IF bIX_TriplexRPMAutoMode = 0 OR bTriplexRPMEnable  = 0 (*Если переключен в режим "Ручной" извне переключателем или отключен с дисплея, то ПИД отключаем*)
THEN
	PID_2_Reset    := 1;
	(*rSet_GN2Rate   := 0;  ЗАЧЕМ!!!!!!!!!!!!!!!!!!!*)
	PID_2_Y_Manual := 1;
ELSE
	PID_2_Reset    := 0;
	PID_2_Y_Manual := 0;
END_IF;

(*-----------------------------------------------------------------------------------------------------------------------------------------------------------------------------------*)
(*Ограничиваем устанавливаемое максимальное значение оборотов*)

IF rSet_TriplexRPM > 975 THEN
	rSet_TriplexRPM := 975;
END_IF;

(*-----------------------------------------------------------------------------------------------------------------------------------------------------------------------------------*)
(*ПИД-контур 1 поддержания скорости НВД*)

PID_2(Actual      := rFRQ_TriplexRPM,
	Set_Point     := rSet_TriplexRPM,
	KP            := rArrayDataPID_P_Coef[2],
	TN            := rArrayDataPID_I_Coef[2],
	TV            := rArrayDataPID_D_Coef[2],
	Y_Manual      := PID_2_Y_Manual,
	Y_Offset      := rArrayDataPID_Shift[2],
	Y_Min         := rArrayDataPWM_YL[2],
	Y_Max         := rArrayDataPWM_YH[2] (*PID_2_Y_Max*),
	Manual        := PID_2_Manual,
	Reset         := PID_2_Reset,
	Y             => rPWM_TriplexRPM,
	Limits_Active => PID_2_Limits,
	Overflow      => PID_2_Overflow);

rArrayDataRAWPID[2] := rPWM_TriplexRPM;

(*-----------------------------------------------------------------------------------------------------------------------------------------------------------------------------------*)
(*Отключаемся от управления ШИМ в режиме "Ручной"*)

IF bIX_TriplexRPMAutoMode = 0 OR bTriplexRPMEnable  = 0 (*Если переключен в режим "Ручной" извне переключателем или отключен с дисплея, то ШИМ отключаем*)
THEN
	rPWM_TriplexRPM := 0;
END_IF;

(*-----------------------------------------------------------------------------------------------------------------------------------------------------------------------------------*)
(*Обработка байта описания канала*)

CASE dwArrayDataPWM_DZ_MIN[2] OF
	0: rPWM_TriplexRPM := rPWM_TriplexRPM;
	1: rPWM_TriplexRPM := rArrayDataPWM_DZ_MAX[2];
	2: rPWM_TriplexRPM := rPWM_TriplexRPM * rArrayDataPWM_DZ_MAX[2];
	ELSE rPWM_TriplexRPM := rPWM_TriplexRPM;
END_CASE;

rArrayDataRAWPWM[2] := rPWM_TriplexRPM;

(*-----------------------------------------------------------------------------------------------------------------------------------------------------------------------------------*)
(*ШИМ-контроллер поддержания скорости НВД*)

TriplexRPMFreqPWM(dwReriodPWM := dwArrayAverTimePWM[2], wFrequencyPWM => , bRestartPWM => );

PWM2(INIT := (bFirstIn OR TriplexRPMFreqPWM.bRestartPWM), FREQUENCY := TriplexRPMFreqPWM.wFrequencyPWM, CHANNEL := 1, VALUE := REAL_TO_WORD(rPWM_TriplexRPM), CHANGE := TRUE, DITHER_VALUE := 10, DITHER_FREQUENCY := 140);

(*-----------------------------------------------------------------------------------------------------------------------------------------------------------------------------------*)
(**)

bIX_TriplexRPMAutoModePrev := bIX_TriplexRPMAutoMode;

(*-----------------------------------------------------------------------------------------------------------------------------------------------------------------------------------*)
(*Расчет рассогласования расчетной и текущей величины*)

rTriplexRPM_Calc := TriplexRPM_calculation(rPWMcurr := (rPWM_TriplexRPM / 10), rRPMeng := DINT_TO_REAL(diCurrentEngineRPM));

IF rFRQ_TriplexRPM > 1
THEN
	rTriplexRPM_Err := (rTriplexRPM_Calc - rFRQ_TriplexRPM) * 100 / rFRQ_TriplexRPM;
ELSE
	rTriplexRPM_Err := 0;
END_IF;

(*-----------------------------------------------------------------------------------------------------------------------------------------------------------------------------------*)
(*bErrorNumber16 - Ошибка 16. НВД. Переведите регулятор в положение «0»*)
(*
IF byCurrStep = 3 AND bTriplexRPMEnable = 1 AND ABS(rTriplexRPM_Err) > 20
THEN
	bErrorNumber16  := 1;(*РАБОТАЕМ С ПРЕДУПРЕЖДЕНИЕМ*)
	dwHornEnable.16 := 0;(*Сирена отключена*)
ELSE
	bErrorNumber16  := 0;
	dwHornEnable.16 := 0;
END_IF;*)
END_PROGRAM

(* POU Service/Temperature_calculation, ST *)
FUNCTION Temperature_calculation : REAL (*Tемпература предварительного прогрева*)

VAR_INPUT
	rTmin : REAL := 0;(*Минимальная температура прогрева, C*)
	rVreq : REAL := 0;(*Заданный расход газообразного азота, м3/мин*)
	rPprs : REAL := 0;(*Давление нагнетания, Мпа*)
	rTreq : REAL := 0;(*Заданная температура нагнетания, С*)
	rK    : REAL := 0;(*Коэффициент теплопередачи*)
END_VAR

VAR
	rTadd : REAL := 0;(*Дополнительная температура подогрева связанная с расходом, C*)
END_VAR
(*-----------------------------------------------------------------------------------------------------------------------------------------------------------------------------------*)
(**)

IF rPprs > 0.1
THEN
	rTadd := 1.8741643E-5 * rVreq * (11760 - 86.5 * SQRT(10 * rPprs - 1) + 0.0255 * (EXPT((rTreq + 273.15), 2) - EXPT(293.15, 2)));
ELSE
	rTadd := 1.8741643E-5 * rVreq * (11760 - 86.5 * SQRT(10 * 0.1 - 1) + 0.0255 * (EXPT((rTreq + 273.15), 2) - EXPT(293.15, 2)));
END_IF;

Temperature_calculation := rTmin + rTadd;
END_FUNCTION

(* POU Service/TriplexRPM_calculation, ST *)
FUNCTION TriplexRPM_calculation : REAL (*Расчетное значение оборотов НВД, об/мин*)

VAR_INPUT
	rPWMcurr : REAL;(*Текущее значение ШИМ, %*)
	rRPMeng  : REAL;(*Обороты двигателя, об/мин*)
END_VAR

VAR
END_VAR
(*-----------------------------------------------------------------------------------------------------------------------------------------------------------------------------------*)
(**)

TriplexRPM_calculation := 0.002187 * rRPMeng * (10 * rPWMcurr - rArrayDataPID_Shift[2]);
END_FUNCTION

(* POU ChannelCalc_processing, ST *)
PROGRAM ChannelCalc_processing

VAR_INPUT
	bInit             : BOOL;
END_VAR

VAR
	AIN_processing_00 : Linearization_AIN_processing;
	AIN_processing_01 : Linearization_AIN_processing;

	AIN_processing_03 : Linearization_AIN_processing;
	AIN_processing_04 : Linearization_AIN_processing;
	AIN_processing_05 : Linearization_AIN_processing;

	AIN_processing_08 : Linearization_AIN_processing;

	PIN_processing_00 : Linearization_PIN_processing;

	PWM_processing_00 : Extraction_PWM_processing;
	PWM_processing_01 : Extraction_PWM_processing;
	PWM_processing_02 : Extraction_PWM_processing;

	PID_processing_00 : Extraction_PID_processing;
	PID_processing_01 : Extraction_PID_processing;
	PID_processing_02 : Extraction_PID_processing;

	i                 : INT := 0;
END_VAR
(*-----------------------------------------------------------------------------------------------------------------------------------------------------------------------------------*)
(**)

FOR i := 0 TO 63 DO

	IF aPage_Channel[i].PARAM_00 = 0
	THEN
		aPage_Channel[i].PARAM_08 := rArrayDataRAWADC[aPage_Channel[i].PARAM_09];
	END_IF;

	IF aPage_Channel[i].PARAM_00 = 1
	THEN
		aPage_Channel[i].PARAM_08 := rArrayDataRAWPIN[aPage_Channel[i].PARAM_09];
	END_IF;

	IF aPage_Channel[i].PARAM_00 = 2
	THEN
		aPage_Channel[i].PARAM_08 := rArrayDataRAWPWM[aPage_Channel[i].PARAM_09];
	END_IF;

	IF aPage_Channel[i].PARAM_00 = 3
	THEN
		aPage_Channel[i].PARAM_08 := rArrayDataRAWPID[aPage_Channel[i].PARAM_09];
	END_IF;

END_FOR;

(*-----------------------------------------------------------------------------------------------------------------------------------------------------------------------------------*)
(**)

AIN_processing_00(
	Page_Channel_AIN := aPage_Channel[0],
	rADC_ValueHigh   := rADC_ValueHigh,
	rADC_ValueLow    := rADC_ValueLow,
	sParamName       => ,
	rOutputValue     => rIW_BoostPres,
	bErrADC_Value    => bErrorBoostPres,
	bErrInputValue   => );

AIN_processing_01(
	Page_Channel_AIN := aPage_Channel[1],
	rADC_ValueHigh   := rADC_ValueHigh,
	rADC_ValueLow    := rADC_ValueLow,
	sParamName       => ,
	rOutputValue     => rIW_LN2_Temp,
	bErrADC_Value    => bErrorLN2_Temp,
	bErrInputValue   => );

AIN_processing_03(
	Page_Channel_AIN := aPage_Channel[2],
	rADC_ValueHigh   := rADC_ValueHigh,
	rADC_ValueLow    := rADC_ValueLow,
	sParamName       => ,
	rOutputValue     => rIW_GN2_Temp,
	bErrADC_Value    => bErrorGN2_Temp,
	bErrInputValue   => );

AIN_processing_04(
	Page_Channel_AIN := aPage_Channel[3],
	rADC_ValueHigh   := rADC_ValueHigh,
	rADC_ValueLow    := rADC_ValueLow,
	sParamName       => ,
	rOutputValue     => rIW_GN2_Pres,
	bErrADC_Value    => bErrorGN2_Pres,
	bErrInputValue   => );

AIN_processing_05(
	Page_Channel_AIN := aPage_Channel[4],
	rADC_ValueHigh   := rADC_ValueHigh,
	rADC_ValueLow    := rADC_ValueLow,
	sParamName       => ,
	rOutputValue     => rIW_HydHeatPres,
	bErrADC_Value    => bErrorHydHeatPres,
	bErrInputValue   => );

AIN_processing_08(
	Page_Channel_AIN := aPage_Channel[5],
	rADC_ValueHigh   := rADC_ValueHigh,
	rADC_ValueLow    := rADC_ValueLow,
	sParamName       => ,
	rOutputValue     => rIW_CoolTempIn,
	bErrADC_Value    => bErrorCoolTempIn,
	bErrInputValue   => );

(*-----------------------------------------------------------------------------------------------------------------------------------------------------------------------------------*)
(**)

PIN_processing_00(
	Page_Channel_PIN := aPage_Channel[6],
	rFRQ_ValueHigh   := 10_000,
	rFRQ_ValueLow    := -1,
	sParamName       => ,
	rOutputValue     => rFRQ_TriplexRPM,
	bErrFRQ_Value    => ,
	bErrInputValue   => );

IF diCurrentEngineRPM < 500
THEN
	rFRQ_TriplexRPM := 0;
END_IF;

(*-----------------------------------------------------------------------------------------------------------------------------------------------------------------------------------*)
(**)

PWM_processing_00(
	Page_Channel_PWM := aPage_Channel[7],
	sParamName       =>,
	rDataPWM_XH      => rArrayDataPWM_XH[1],
	rDataPWM_XL      => rArrayDataPWM_XL[1],
	rDataPWM_YH      => rArrayDataPWM_YH[1],
	rDataPWM_YL      => rArrayDataPWM_YL[1],
	dwAverTimePWM    => dwArrayAverTimePWM[1],
	rDataPWM_DZ_MAX  => rArrayDataPWM_DZ_MAX[1],
	dwDataPWM_DZ_MIN => dwArrayDataPWM_DZ_MIN[1],
	dwNumberPWM      => dwArrayNumberPWM[1],
	rParam10PWM      => rArrayParam10PWM[1]);

PWM_processing_01(
	Page_Channel_PWM := aPage_Channel[8],
	sParamName       =>,
	rDataPWM_XH      => rArrayDataPWM_XH[2],
	rDataPWM_XL      => rArrayDataPWM_XL[2],
	rDataPWM_YH      => rArrayDataPWM_YH[2],
	rDataPWM_YL      => rArrayDataPWM_YL[2],
	dwAverTimePWM    => dwArrayAverTimePWM[2],
	rDataPWM_DZ_MAX  => rArrayDataPWM_DZ_MAX[2],
	dwDataPWM_DZ_MIN => dwArrayDataPWM_DZ_MIN[2],
	dwNumberPWM      => dwArrayNumberPWM[2],
	rParam10PWM      => rArrayParam10PWM[2]);

PWM_processing_02(
	Page_Channel_PWM := aPage_Channel[9],
	sParamName       =>,
	rDataPWM_XH      => rArrayDataPWM_XH[3],
	rDataPWM_XL      => rArrayDataPWM_XL[3],
	rDataPWM_YH      => rArrayDataPWM_YH[3],
	rDataPWM_YL      => rArrayDataPWM_YL[3],
	dwAverTimePWM    => dwArrayAverTimePWM[3],
	rDataPWM_DZ_MAX  => rArrayDataPWM_DZ_MAX[3],
	dwDataPWM_DZ_MIN => dwArrayDataPWM_DZ_MIN[3],
	dwNumberPWM      => dwArrayNumberPWM[3],
	rParam10PWM      => rArrayParam10PWM[3]);

(*-----------------------------------------------------------------------------------------------------------------------------------------------------------------------------------*)
(**)

PID_processing_00(
	Page_Channel_PID := aPage_Channel[10],
	sParamName       =>,
	rDataPID_P_Coef  => rArrayDataPID_P_Coef[1],
	rDataPID_I_Coef  => rArrayDataPID_I_Coef[1],
	rDataPID_D_Coef  => rArrayDataPID_D_Coef[1],
	rDataPID_Shift   => rArrayDataPID_Shift[1],
	dwAverTimePID    => dwArrayAverTimePID[1],
	rCoeffPID        => rArrayCoeffPID[1],
	dwDescriptPID    => dwArrayDescriptPID[1],
	dwNumberPID      => dwArrayNumberPID[1],
	rParam10PID      => rArrayParam10PID[1]);

PID_processing_01(
	Page_Channel_PID := aPage_Channel[11],
	sParamName       =>,
	rDataPID_P_Coef  => rArrayDataPID_P_Coef[2],
	rDataPID_I_Coef  => rArrayDataPID_I_Coef[2],
	rDataPID_D_Coef  => rArrayDataPID_D_Coef[2],
	rDataPID_Shift   => rArrayDataPID_Shift[2],
	dwAverTimePID    => dwArrayAverTimePID[2],
	rCoeffPID        => rArrayCoeffPID[2],
	dwDescriptPID    => dwArrayDescriptPID[2],
	dwNumberPID      => dwArrayNumberPID[2],
	rParam10PID      => rArrayParam10PID[2]);

PID_processing_02(
	Page_Channel_PID := aPage_Channel[12],
	sParamName       =>,
	rDataPID_P_Coef  => rArrayDataPID_P_Coef[3],
	rDataPID_I_Coef  => rArrayDataPID_I_Coef[3],
	rDataPID_D_Coef  => rArrayDataPID_D_Coef[3],
	rDataPID_Shift   => rArrayDataPID_Shift[3],
	dwAverTimePID    => dwArrayAverTimePID[3],
	rCoeffPID        => rArrayCoeffPID[3],
	dwDescriptPID    => dwArrayDescriptPID[3],
	dwNumberPID      => dwArrayNumberPID[3],
	rParam10PID      => rArrayParam10PID[3]);

(*-----------------------------------------------------------------------------------------------------------------------------------------------------------------------------------*)
(**)

bCommomErrorADC := (bErrorBoostPres OR
					bErrorLN2_Temp OR
					bErrorGN2_Temp OR
					bErrorGN2_Pres OR
					(*bErrorHydHeatPres OR*)
					bErrorCoolTempIn);

(*-----------------------------------------------------------------------------------------------------------------------------------------------------------------------------------*)
(*Расчет текущей производительности установки*)

IF rFRQ_TriplexRPM > 0
THEN
	rCurrent_GN2Rate := 0.08786324786325 * rFRQ_TriplexRPM; (*м3/оборот * оборот/мин*)
ELSE
	rCurrent_GN2Rate := 0;
END_IF;

udiCurrent_GN2RateLitres := REAL_TO_DWORD(rCurrent_GN2Rate * 1000);

(*-----------------------------------------------------------------------------------------------------------------------------------------------------------------------------------*)
(**)
END_PROGRAM

(* POU Linearization_AIN_processing, ST *)
FUNCTION_BLOCK Linearization_AIN_processing

VAR_INPUT
	Page_Channel_AIN  : Page_Channel;
	rADC_ValueHigh    : REAL;
	rADC_ValueLow     : REAL;
END_VAR

VAR_OUTPUT
	sParamName        : STRING(32);
	rOutputValue      : REAL := 0;
	bErrADC_Value     : BOOL := 0;
	bErrInputValue    : BOOL := 0;
END_VAR

VAR
	rArrayDataADC     : ARRAY [0..257] OF REAL;(*Массив необработанных данных канала, REAL*)
	rTotalADC         : REAL := 0;(**)
	iIndexReadings    : INT  := 0;(**)
	diNumReadings     : DINT := 10;(*Рассчитанное число измерений для усреднения*)
	diNumReadingsPrev : DINT := 0;
	rDataOutADC       : REAL;(*Усредненное значение канала*)
	i                 : INT  := 0;

	bErrADC_ValueHigh : BOOL := 0;
	bErrADC_ValueLow  : BOOL := 0;
END_VAR
(*-----------------------------------------------------------------------------------------------------------------------------------------------------------------------------------*)
(**)

sParamName := Page_Channel_AIN.PARAM_NAME;

(*-----------------------------------------------------------------------------------------------------------------------------------------------------------------------------------*)
(*Усредняем значене канала*)

diNumReadings := (DWORD_TO_DINT(Page_Channel_AIN.PARAM_05) * 1000) / 10_000 (*DWORD_TO_DINT(dwCycleTime)*);(**)
IF diNumReadings < 1   THEN diNumReadings := 1;   END_IF;
IF diNumReadings > 255 THEN diNumReadings := 255; END_IF;

IF diNumReadings <> diNumReadingsPrev
THEN
	rTotalADC := 0;
	FOR i := 1 TO DINT_TO_INT(diNumReadings) DO
	rTotalADC := rTotalADC + rArrayDataADC[i - 1];
	END_FOR;
END_IF;

diNumReadingsPrev := diNumReadings;

rTotalADC := rTotalADC - rArrayDataADC[iIndexReadings];(*subtract the last reading*)

rArrayDataADC[iIndexReadings] := Page_Channel_AIN.PARAM_08;(*read from the sensor*)

rTotalADC := rTotalADC + rArrayDataADC[iIndexReadings];(*add the reading to the total*)

iIndexReadings := iIndexReadings + 1;(*advance to the next position in the array*)

IF INT_TO_DINT(iIndexReadings) >= diNumReadings THEN iIndexReadings := 0; END_IF;(*if we're at the end of the array... ...wrap around to the beginning*)

rDataOutADC := rTotalADC / DINT_TO_REAL(diNumReadings);(**)

(*-----------------------------------------------------------------------------------------------------------------------------------------------------------------------------------*)
(*Основная обработка аналогового канала*)

(*Обработка обрывов (значение меньше минимально допустимого) и КЗ (значение больше максимально допустимого) по входу канала*)
IF rDataOutADC > rADC_ValueHigh
THEN bErrADC_ValueHigh := 1;
ELSE bErrADC_ValueHigh := 0;
END_IF;

IF rDataOutADC < rADC_ValueLow
THEN bErrADC_ValueLow := 1;
ELSE bErrADC_ValueLow := 0;
END_IF;

bErrADC_Value := bErrADC_ValueHigh OR bErrADC_ValueLow;

(*Масштабирование значений каналов*)
IF Page_Channel_AIN.PARAM_01 = Page_Channel_AIN.PARAM_02
THEN
	rOutputValue := rDataOutADC;(*Защита от деления на 0, выводим необработанные значения АЦП*)
	bErrInputValue := 1;
ELSE
	rOutputValue := (Page_Channel_AIN.PARAM_03 - Page_Channel_AIN.PARAM_04) / (Page_Channel_AIN.PARAM_01 - Page_Channel_AIN.PARAM_02) * rDataOutADC + (Page_Channel_AIN.PARAM_04 - (Page_Channel_AIN.PARAM_03 - Page_Channel_AIN.PARAM_04) / (Page_Channel_AIN.PARAM_01 - Page_Channel_AIN.PARAM_02) * Page_Channel_AIN.PARAM_02);
	bErrInputValue := 0;
END_IF;

(*Обработка байта описания канала*)
CASE Page_Channel_AIN.PARAM_07 OF
	0: rOutputValue := rOutputValue;
	1: rOutputValue := Page_Channel_AIN.PARAM_06;
	2: rOutputValue := rOutputValue * Page_Channel_AIN.PARAM_06;
ELSE
	rOutputValue := rOutputValue;
END_CASE;

(*Если обнаружена ошибка по каналу, то подставляем заведомо неверное число*)
	IF bErrADC_Value = 1 OR bErrInputValue = 1 THEN rOutputValue := -9999; END_IF;

(*-----------------------------------------------------------------------------------------------------------------------------------------------------------------------------------*)
(**)
END_FUNCTION_BLOCK

(* POU Linearization_PIN_processing, ST *)
FUNCTION_BLOCK Linearization_PIN_processing

VAR_INPUT
	Page_Channel_PIN  : Page_Channel;
	rFRQ_ValueHigh    : REAL;
	rFRQ_ValueLow     : REAL;
END_VAR

VAR_OUTPUT
	sParamName        : STRING(32);
	rOutputValue      : REAL := 0;
	bErrFRQ_Value     : BOOL := 0;
	bErrInputValue    : BOOL := 0;
END_VAR

VAR
	rArrayDataFRQ     : ARRAY [0..257] OF REAL;(*Массив необработанных данных канала, REAL*)
	rTotalFRQ         : REAL := 0;(**)
	rTotalFRQ2        : REAL := 0;(**)
	iIndexReadings    : INT  := 0;(**)
	diNumReadings     : DINT := 10;(*Рассчитанное число измерений для усреднения*)
	diNumReadingsPrev : DINT := 0;
	rDataOutFRQ       : REAL;(*Усредненное значение канала*)
	i                 : INT  := 0;

	bErrFRQ_ValueHigh : BOOL := 0;
	bErrFRQ_ValueLow  : BOOL := 0;
END_VAR
(*-----------------------------------------------------------------------------------------------------------------------------------------------------------------------------------*)
(**)

sParamName := Page_Channel_PIN.PARAM_NAME;

(*-----------------------------------------------------------------------------------------------------------------------------------------------------------------------------------*)
(*Усредняем значене канала*)

diNumReadings := (DWORD_TO_DINT(Page_Channel_PIN.PARAM_05) * 1000) / 10_000 (*DWORD_TO_DINT(dwCycleTime)*);(**)
IF diNumReadings < 1   THEN diNumReadings := 1;   END_IF;
IF diNumReadings > 255 THEN diNumReadings := 255; END_IF;

IF diNumReadings <> diNumReadingsPrev
THEN
	rTotalFRQ  := 0;
	rTotalFRQ2 := 0;
	FOR i := 1 TO DINT_TO_INT(diNumReadings) DO
	rTotalFRQ  := rTotalFRQ  + rArrayDataFRQ[i - 1];
	rTotalFRQ2 := rTotalFRQ;
	END_FOR;
END_IF;

diNumReadingsPrev := diNumReadings;

rTotalFRQ := rTotalFRQ - rArrayDataFRQ[iIndexReadings];(*subtract the last reading*)

rArrayDataFRQ[iIndexReadings] := Page_Channel_PIN.PARAM_08;(*read from the sensor*)

rTotalFRQ := rTotalFRQ + rArrayDataFRQ[iIndexReadings];(*add the reading to the total*)

rTotalFRQ2 := rTotalFRQ2 + rArrayDataFRQ[iIndexReadings];

iIndexReadings := iIndexReadings + 1;(*advance to the next position in the array*)

IF INT_TO_DINT(iIndexReadings) >= diNumReadings
THEN
	IF rTotalFRQ2 < 1
	THEN rTotalFRQ := 0;
	END_IF;
END_IF;

IF INT_TO_DINT(iIndexReadings) >= diNumReadings THEN iIndexReadings := 0; rTotalFRQ2 := 0; END_IF;(*if we're at the end of the array... ...wrap around to the beginning*)

rDataOutFRQ := rTotalFRQ / DINT_TO_REAL(diNumReadings);(**)

(*-----------------------------------------------------------------------------------------------------------------------------------------------------------------------------------*)
(*Основная обработка частотного канала*)

(*Обработка ошибочных частот (значение меньше минимально допустимого и значение больше максимально допустимого) по входу канала*)
IF rDataOutFRQ > rFRQ_ValueHigh
THEN bErrFRQ_ValueHigh := 1;
ELSE bErrFRQ_ValueHigh := 0;
END_IF;

IF rDataOutFRQ < rFRQ_ValueLow
THEN bErrFRQ_ValueLow := 1;
ELSE bErrFRQ_ValueLow := 0;
END_IF;

bErrFRQ_Value := bErrFRQ_ValueHigh OR bErrFRQ_ValueLow;

(*Масштабирование значений каналов*)
IF Page_Channel_PIN.PARAM_01 = Page_Channel_PIN.PARAM_02
THEN
	rOutputValue := rDataOutFRQ;(*Защита от деления на 0, выводим необработанные значения частоты*)
	bErrInputValue := 1;
ELSE
	rOutputValue := (Page_Channel_PIN.PARAM_03 - Page_Channel_PIN.PARAM_04) / (Page_Channel_PIN.PARAM_01 - Page_Channel_PIN.PARAM_02) * rDataOutFRQ;
	bErrInputValue := 0;
END_IF;

(*Обработка байта описания канала*)
CASE Page_Channel_PIN.PARAM_07 OF
	0: rOutputValue := rOutputValue;
	1: rOutputValue := Page_Channel_PIN.PARAM_06;
	2: rOutputValue := rOutputValue * Page_Channel_PIN.PARAM_06;
ELSE
	rOutputValue := rOutputValue;
END_CASE;

(*Если обнаружена ошибка по каналу, то подставляем заведомо неверное число*)
	IF bErrFRQ_Value = 1 OR bErrInputValue = 1 THEN rOutputValue := -9999; END_IF;

(*-----------------------------------------------------------------------------------------------------------------------------------------------------------------------------------*)
(**)
END_FUNCTION_BLOCK

(* POU Extraction_PWM_processing, ST *)
FUNCTION_BLOCK Extraction_PWM_processing

VAR_INPUT
	Page_Channel_PWM : Page_Channel;
END_VAR

VAR_OUTPUT
	sParamName       : STRING(32);
	rDataPWM_XH      : REAL;
	rDataPWM_XL      : REAL;
	rDataPWM_YH      : REAL;
	rDataPWM_YL      : REAL;
	dwAverTimePWM    : DWORD;
	rDataPWM_DZ_MAX  : REAL;
	dwDataPWM_DZ_MIN : DWORD;
	dwNumberPWM      : DWORD;
	rParam10PWM      : REAL;
END_VAR

VAR
END_VAR
(*-----------------------------------------------------------------------------------------------------------------------------------------------------------------------------------*)
(**)

sParamName       := Page_Channel_PWM.PARAM_NAME;
rDataPWM_XH      := Page_Channel_PWM.PARAM_01;
rDataPWM_XL      := Page_Channel_PWM.PARAM_02;
rDataPWM_YH      := Page_Channel_PWM.PARAM_03;
rDataPWM_YL      := Page_Channel_PWM.PARAM_04;
dwAverTimePWM    := Page_Channel_PWM.PARAM_05;
rDataPWM_DZ_MAX  := Page_Channel_PWM.PARAM_06;
dwDataPWM_DZ_MIN := Page_Channel_PWM.PARAM_07;

dwNumberPWM      := Page_Channel_PWM.PARAM_09;
rParam10PWM      := Page_Channel_PWM.PARAM_10;
END_FUNCTION_BLOCK

(* POU Extraction_PID_processing, ST *)
FUNCTION_BLOCK Extraction_PID_processing

VAR_INPUT
	Page_Channel_PID : Page_Channel;
END_VAR

VAR_OUTPUT
	sParamName      : STRING(32);
	rDataPID_P_Coef : REAL;
	rDataPID_I_Coef : REAL;
	rDataPID_D_Coef : REAL;
	rDataPID_Shift  : REAL;
	dwAverTimePID   : DWORD;
	rCoeffPID       : REAL;
	dwDescriptPID   : DWORD;
	dwNumberPID     : DWORD;
	rParam10PID     : REAL;
END_VAR

VAR
END_VAR
(*-----------------------------------------------------------------------------------------------------------------------------------------------------------------------------------*)
(**)

sParamName      := Page_Channel_PID.PARAM_NAME;
rDataPID_P_Coef := Page_Channel_PID.PARAM_01;
rDataPID_I_Coef := Page_Channel_PID.PARAM_02;
rDataPID_D_Coef := Page_Channel_PID.PARAM_03;
rDataPID_Shift  := Page_Channel_PID.PARAM_04;
dwAverTimePID   := Page_Channel_PID.PARAM_05;
rCoeffPID       := Page_Channel_PID.PARAM_06;
dwDescriptPID   := Page_Channel_PID.PARAM_07;

dwNumberPID     := Page_Channel_PID.PARAM_09;
rParam10PID     := Page_Channel_PID.PARAM_10;
END_FUNCTION_BLOCK

(* POU Adder_processing, ST *)
PROGRAM Adder_processing

VAR_INPUT
	bInit                    : BOOL;
END_VAR

VAR
	dwTimePrevious           : DWORD := 0;
	dwDeltaTime              : DWORD := 0;

	instFRAMWrite            : FRAMWRITE;
	instFRAMRead             : FRAMREAD;

	i                        : INT;
	k                        : INT;
END_VAR
(*-----------------------------------------------------------------------------------------------------------------------------------------------------------------------------------*)
(*Собираем флаги сброса сумматоров частотных каналов в массив*)

bArrayDataPINAdderReset[1] := bResetTotalAmountGN2 (*bFlowmeterReset_1*);
bArrayDataPINAdderReset[2] := bFlowmeterReset_2;
bArrayDataPINAdderReset[3] := bFlowmeterReset_3;
bArrayDataPINAdderReset[4] := bFlowmeterReset_4;

(*-----------------------------------------------------------------------------------------------------------------------------------------------------------------------------------*)
(*Накопление текущих значений и обработка флагов сброса суммирующих каналов*)

IF k < 100 (*10?*) THEN k := k + 1; ELSE k := 0; END_IF;

IF k = 1
THEN
	dwDeltaTime := (dwTime_US - dwTimePrevious) / 1000;
	FOR i := 1 TO 4 DO
		instFRAMRead(Enable := TRUE, SRC := iMemAdrPINAdder[i], LEN := 4, DST := ADR(udiArrayDataPINAdderOut[i]));(*Извлечение из FRAM значение расходомера i*)

		IF bArrayDataPINAdderReset[i] = 1
			THEN udiArrayDataPINAdderOut[i] := 0;
			ELSE udiArrayDataPINAdderOut[i] := udiArrayDataPINAdderOut[i] + ((udiCurrent_GN2RateLitres * 10 * DWORD_TO_UDINT(dwDeltaTime)) / 60 / 1_000);(*Храним в 0,1 литра*)
		END_IF;

		instFRAMWrite(Enable := TRUE, DST := iMemAdrPINAdder[i], LEN := 4, SRC := ADR(udiArrayDataPINAdderOut[i])); (*Cохранение в FRAM значение расходомера i*)
		END_FOR;

	dwTimePrevious := dwTime_US;

(*-----------------------------------------------------------------------------------------------------------------------------------------------------------------------------------*)
(*Сброс флага "Обнулить накопленное значение расходомера"*)

	bResetTotalAmountGN2 (*bFlowmeterReset_1*) := 0;(*Сброс флага "Обнулить накопленное значение расходомера 0"*)
	bFlowmeterReset_2 := 0;(*Сброс флага "Обнулить накопленное значение расходомера 1"*)
	bFlowmeterReset_3 := 0;(*Сброс флага "Обнулить накопленное значение расходомера 2"*)
	bFlowmeterReset_4 := 0;(*Сброс флага "Обнулить накопленное значение расходомера 3"*)
END_IF;

(*-----------------------------------------------------------------------------------------------------------------------------------------------------------------------------------*)
(*Оформляем необходимые данные для дальнейшей обработки в других блоках*)

rTotalAmountGN2 := UDINT_TO_REAL(udiArrayDataPINAdderOut[1]) / 1000 / 10;
END_PROGRAM

(* POU Output Modules/ProcessState_processing, ST *)
PROGRAM ProcessState_processing

VAR_INPUT
	bFirstIn   : BOOL;
END_VAR

VAR
END_VAR
dwProcessState := 16#0000;

dwProcessState.0 := bDefaultSettings;
dwProcessState.1 := bStop;
dwProcessState.2 := bHornDisable;
dwProcessState.3 := bBlockDisable;

dwProcessState.5 := bIX_BlockOff;

dwProcessState.7 := NOT bQX_TriplexEmergStopTrig;
END_PROGRAM

(* POU Output Modules/Error_processing, ST *)
PROGRAM Error_processing

VAR_INPUT
	bFirstIn            : BOOL;
END_VAR

VAR
	RSInst              : RS;(*Триггер на блокировку*)

	RTRIGInst01         : R_TRIG;
	RTRIGInst02         : R_TRIG;
	RTRIGInst03         : R_TRIG;
	RTRIGInst04         : R_TRIG;
	RTRIGInst05         : R_TRIG;
	RTRIGInst06         : R_TRIG;
	RTRIGInst07         : R_TRIG;
	RTRIGInst08         : R_TRIG;
	RTRIGInst09         : R_TRIG;
	RTRIGInst10         : R_TRIG;
	RTRIGInst11         : R_TRIG;
	RTRIGInst12         : R_TRIG;
	RTRIGInst13         : R_TRIG;
	RTRIGInst14         : R_TRIG;
	RTRIGInst15         : R_TRIG;
	RTRIGInst16         : R_TRIG;

	RTRIGInst17         : R_TRIG;
	RTRIGInst18         : R_TRIG;
	RTRIGInst19         : R_TRIG;
	RTRIGInst20         : R_TRIG;
	RTRIGInst21         : R_TRIG;
	RTRIGInst22         : R_TRIG;
	RTRIGInst23         : R_TRIG;
	RTRIGInst24         : R_TRIG;
	RTRIGInst25         : R_TRIG;
	RTRIGInst26         : R_TRIG;
	RTRIGInst27         : R_TRIG;
	RTRIGInst28         : R_TRIG;
	RTRIGInst29         : R_TRIG;
	RTRIGInst30         : R_TRIG;
	RTRIGInst31         : R_TRIG;
	RTRIGInst32         : R_TRIG;

	bErrorNumber01RTrig : BOOL := 0;
	bErrorNumber02RTrig : BOOL := 0;
	bErrorNumber03RTrig : BOOL := 0;
	bErrorNumber04RTrig : BOOL := 0;
	bErrorNumber05RTrig : BOOL := 0;
	bErrorNumber06RTrig : BOOL := 0;
	bErrorNumber07RTrig : BOOL := 0;
	bErrorNumber08RTrig : BOOL := 0;
	bErrorNumber09RTrig : BOOL := 0;
	bErrorNumber10RTrig : BOOL := 0;
	bErrorNumber11RTrig : BOOL := 0;
	bErrorNumber12RTrig : BOOL := 0;
	bErrorNumber13RTrig : BOOL := 0;
	bErrorNumber14RTrig : BOOL := 0;
	bErrorNumber15RTrig : BOOL := 0;
	bErrorNumber16RTrig : BOOL := 0;

	bErrorNumber17RTrig : BOOL := 0;
	bErrorNumber18RTrig : BOOL := 0;
	bErrorNumber19RTrig : BOOL := 0;
	bErrorNumber20RTrig : BOOL := 0;
	bErrorNumber21RTrig : BOOL := 0;
	bErrorNumber22RTrig : BOOL := 0;
	bErrorNumber23RTrig : BOOL := 0;
	bErrorNumber24RTrig : BOOL := 0;
	bErrorNumber25RTrig : BOOL := 0;
	bErrorNumber26RTrig : BOOL := 0;
	bErrorNumber27RTrig : BOOL := 0;
	bErrorNumber28RTrig : BOOL := 0;
	bErrorNumber29RTrig : BOOL := 0;
	bErrorNumber30RTrig : BOOL := 0;
	bErrorNumber31RTrig : BOOL := 0;
	bErrorNumber32RTrig : BOOL := 0;

	RSInst01            : RS;
	RSInst02            : RS;
	RSInst03            : RS;
	RSInst04            : RS;
	RSInst05            : RS;
	RSInst06            : RS;
	RSInst07            : RS;
	RSInst08            : RS;
	RSInst09            : RS;
	RSInst10            : RS;
	RSInst11            : RS;
	RSInst12            : RS;
	RSInst13            : RS;
	RSInst14            : RS;
	RSInst15            : RS;
	RSInst16            : RS;

	RSInst17            : RS;
	RSInst18            : RS;
	RSInst19            : RS;
	RSInst20            : RS;
	RSInst21            : RS;
	RSInst22            : RS;
	RSInst23            : RS;
	RSInst24            : RS;
	RSInst25            : RS;
	RSInst26            : RS;
	RSInst27            : RS;
	RSInst28            : RS;
	RSInst29            : RS;
	RSInst30            : RS;
	RSInst31            : RS;
	RSInst32            : RS;

	bErrorNumber01Trig  : BOOL := 0;
	bErrorNumber02Trig  : BOOL := 0;
	bErrorNumber03Trig  : BOOL := 0;
	bErrorNumber04Trig  : BOOL := 0;
	bErrorNumber05Trig  : BOOL := 0;
	bErrorNumber06Trig  : BOOL := 0;
	bErrorNumber07Trig  : BOOL := 0;
	bErrorNumber08Trig  : BOOL := 0;
	bErrorNumber09Trig  : BOOL := 0;
	bErrorNumber10Trig  : BOOL := 0;
	bErrorNumber11Trig  : BOOL := 0;
	bErrorNumber12Trig  : BOOL := 0;
	bErrorNumber13Trig  : BOOL := 0;
	bErrorNumber14Trig  : BOOL := 0;
	bErrorNumber15Trig  : BOOL := 0;
	bErrorNumber16Trig  : BOOL := 0;

	bErrorNumber17Trig  : BOOL := 0;
	bErrorNumber18Trig  : BOOL := 0;
	bErrorNumber19Trig  : BOOL := 0;
	bErrorNumber20Trig  : BOOL := 0;
	bErrorNumber21Trig  : BOOL := 0;
	bErrorNumber22Trig  : BOOL := 0;
	bErrorNumber23Trig  : BOOL := 0;
	bErrorNumber24Trig  : BOOL := 0;
	bErrorNumber25Trig  : BOOL := 0;
	bErrorNumber26Trig  : BOOL := 0;
	bErrorNumber27Trig  : BOOL := 0;
	bErrorNumber28Trig  : BOOL := 0;
	bErrorNumber29Trig  : BOOL := 0;
	bErrorNumber30Trig  : BOOL := 0;
	bErrorNumber31Trig  : BOOL := 0;
	bErrorNumber32Trig  : BOOL := 0;
END_VAR
(*-----------------------------------------------------------------------------------------------------------------------------------------------------------------------------------*)
(*bErrorNumber01 - Ошибка 01. Нет связи с компьютерной панелью*)

IF bCAN1_J1939NotActive = 1 OR bCAN1_J1939Errors = 1
THEN
	bErrorNumber01 := 1;(*РАБОТАЕМ С ПРЕДУПРЕЖДЕНИЕМ*)
	dwHornEnable.1 := 0;(*Сирена отключена*)
ELSE
	bErrorNumber01 := 0;
	dwHornEnable.1 := 0;
END_IF;

(*-----------------------------------------------------------------------------------------------------------------------------------------------------------------------------------*)
(*bErrorNumber02 - Ошибка 02. Температура газообр. азота ниже допустимого*)

IF rIW_GN2_Temp < -50 AND byCurrStep = 3
THEN
	bErrorNumber02 := 1;(*РАБОТАЕМ С ПРЕДУПРЕЖДЕНИЕМ*)
	dwHornEnable.2 := 0;(*Сирена отключена*)
ELSE
	bErrorNumber02 := 0;
	dwHornEnable.2 := 0;
END_IF;

(*-----------------------------------------------------------------------------------------------------------------------------------------------------------------------------------*)
(*bErrorNumber03 - Ошибка 03. Температура газообр. азота выше допустимого*)

IF rIW_GN2_Temp > 250 AND byCurrStep = 3
THEN
	bErrorNumber03 := 1;(*РАБОТАЕМ С ПРЕДУПРЕЖДЕНИЕМ*)
	dwHornEnable.3 := 0;(*Сирена отключена*)
ELSE
	bErrorNumber03 := 0;
	dwHornEnable.3 := 0;
END_IF;

(*-----------------------------------------------------------------------------------------------------------------------------------------------------------------------------------*)
(*bErrorNumber05 - Ошибка 05. Двигатель. Аварийная остановка*)

IF byCurrStep = 3 AND bIX_EngineStopped = 1
THEN
	bErrorNumber05 := 1;
	bStart := 0;(*ОСТАНОВ И УХОДИМ НА НАЧАЛО*)
(*ELSE
	bErrorNumber05 := 0;*) (*Сброс флага при повторном старте системы*)
END_IF;

(*-----------------------------------------------------------------------------------------------------------------------------------------------------------------------------------*)
(*bErrorNumber06 - Ошибка 06. Двигатель. Обороты «0»*)

IF diCurrentEngineRPM < 100 AND byCurrStep = 3
THEN
	bErrorNumber06 := 1;
	bStart := 0;(*ОСТАНОВ И УХОДИМ НА НАЧАЛО*)
(*ELSE
	bErrorNumber06 := 0;*) (*Сброс флага при повторном старте системы*)
END_IF;

(*-----------------------------------------------------------------------------------------------------------------------------------------------------------------------------------*)
(*bErrorNumber07 - Ошибка 07. НВД. Режим охлаждения (до 20 об/мин )*)

IF bBlockDisable = 1
THEN
	bErrorNumber07 := 1;(*РАБОТАЕМ С ПРЕДУПРЕЖДЕНИЕМ*)
	dwHornEnable.7 := 0;(*Сирена отключена*)
ELSE
	bErrorNumber07 := 0;
	dwHornEnable.7 := 0;
END_IF;

(*-----------------------------------------------------------------------------------------------------------------------------------------------------------------------------------*)
(*bErrorNumber10 - Ошибка 10. Центробеж. насос. Перевести в «Ручной»*)

IF (byCurrStep = 0 OR byCurrStep = 1 OR byCurrStep = 2) AND bIX_BoostPresAutoMode = 1
THEN
	bErrorNumber10         := 1;(*РАБОТАЕМ С ПРЕДУПРЕЖДЕНИЕМ. ИНИЦИАЛИЗАЦИЯ*)
	dwHornEnable.10        := 0;(*Сирена отключена*)
	bQX_EngineStarterBlock := 1;(*Блокируем запуск двигателя, если тумблер в "Авто"*)
ELSE
	bErrorNumber10         := 0;
	dwHornEnable.10        := 0;
END_IF;

(*-----------------------------------------------------------------------------------------------------------------------------------------------------------------------------------*)
(*bErrorNumber11 - Ошибка 11. НВД. Перевести в «Ручной»*)

IF (byCurrStep = 0 OR byCurrStep = 1 OR byCurrStep = 2) AND bIX_TriplexRPMAutoMode = 1
THEN
	bErrorNumber11         := 1;(*РАБОТАЕМ С ПРЕДУПРЕЖДЕНИЕМ. ИНИЦИАЛИЗАЦИЯ*)
	dwHornEnable.11        := 0;(*Сирена отключена*)
	bQX_EngineStarterBlock := 1;(*Блокируем запуск двигателя, если тумблер в "Авто"*)
ELSE
	bErrorNumber11         := 0;
	dwHornEnable.11        := 0;
END_IF;

(*-----------------------------------------------------------------------------------------------------------------------------------------------------------------------------------*)
(*bErrorNumber12 - Ошибка 12. Гидронагрев. Перевести в «Ручной»*)

IF (byCurrStep = 0 OR byCurrStep = 1 OR byCurrStep = 2) AND bIX_HydHeatPresAutoMode = 1
THEN
	bErrorNumber12         := 1;(*РАБОТАЕМ С ПРЕДУПРЕЖДЕНИЕМ. ИНИЦИАЛИЗАЦИЯ*)
	dwHornEnable.12        := 0;(*Сирена отключена*)
	bQX_EngineStarterBlock := 1;(*Блокируем запуск двигателя, если тумблер в "Авто"*)
ELSE
	bErrorNumber12         := 0;
	dwHornEnable.12        := 0;
END_IF;

(*-----------------------------------------------------------------------------------------------------------------------------------------------------------------------------------*)
(*bErrorNumber24 - Ошибка 24. Регуляторы в положении «0»*)

IF (byCurrStep = 0 OR byCurrStep = 1 OR byCurrStep = 2) AND (bIX_TriplexRPMAutoMode = 0 OR bIX_HydHeatPresAutoMode = 0 OR bIX_BoostPresAutoMode = 0)
THEN
	bErrorNumber24  := 1;(*РАБОТАЕМ С ПРЕДУПРЕЖДЕНИЕМ*)
	dwHornEnable.24 := 0;(*Сирена отключена*)
ELSE
	bErrorNumber24  := 0;
	dwHornEnable.24 := 0;
END_IF;

(*-----------------------------------------------------------------------------------------------------------------------------------------------------------------------------------*)
(*bErrorNumber25 - Ошибка 25. Аварийная работа*)

IF bIX_BlockOff = 1
THEN
	bErrorNumber25  := 1;(*РАБОТАЕМ С ПРЕДУПРЕЖДЕНИЕМ*)
	dwHornEnable.25 := 1;(*Сирена включена*)
ELSE
	bErrorNumber25  := 0;
	dwHornEnable.25 := 0;
END_IF;

(*-----------------------------------------------------------------------------------------------------------------------------------------------------------------------------------*)
(*bErrorNumber27 - Ошибка 27. Ошибка CAN2 J1939*)

IF bCAN2_J1939Errors = 1
THEN
	bErrorNumber27  := 0;(*РАБОТАЕМ С ПРЕДУПРЕЖДЕНИЕМ*)
	dwHornEnable.27 := 0;(*Сирена отключена*)
ELSE
	bErrorNumber27  := 0;
	dwHornEnable.27 := 0;
END_IF;

(*-----------------------------------------------------------------------------------------------------------------------------------------------------------------------------------*)
(*bErrorNumber28 - Ошибка 28. Отсутсвует CAN2 J1939*)

IF bCAN2_J1939NotActive = 1
THEN
	bErrorNumber28  := 1;(*РАБОТАЕМ С ПРЕДУПРЕЖДЕНИЕМ*)
	dwHornEnable.28 := 0;(*Сирена отключена*)
ELSE
	bErrorNumber28  := 0;
	dwHornEnable.28 := 0;
END_IF;

(*-----------------------------------------------------------------------------------------------------------------------------------------------------------------------------------*)
(**)

dwErrorState := 0;

(*Собираем в слово 1 состояния ошибок*)
 dwErrorState.0 := bErrorNumber01;
 dwErrorState.1 := bErrorNumber02;
 dwErrorState.2 := bErrorNumber03;
 dwErrorState.3 := bErrorNumber04;
 dwErrorState.4 := bErrorNumber05;
 dwErrorState.5 := bErrorNumber06;
 dwErrorState.6 := bErrorNumber07;
 dwErrorState.7 := bErrorNumber08;

 dwErrorState.8 := bErrorNumber09;
 dwErrorState.9 := bErrorNumber10;
dwErrorState.10 := bErrorNumber11;
dwErrorState.11 := bErrorNumber12;
dwErrorState.12 := bErrorNumber13;
dwErrorState.13 := bErrorNumber14;
dwErrorState.14 := bErrorNumber15;
dwErrorState.15 := bErrorNumber16;

dwErrorState.16 := bErrorNumber17;
dwErrorState.17 := bErrorNumber18;
dwErrorState.18 := bErrorNumber19;
dwErrorState.19 := bErrorNumber20;
dwErrorState.20 := bErrorNumber21;
dwErrorState.21 := bErrorNumber22;
dwErrorState.22 := bErrorNumber23;
dwErrorState.23 := bErrorNumber24;

dwErrorState.24 := bErrorNumber25;
dwErrorState.25 := bErrorNumber26;
dwErrorState.26 := bErrorNumber27;
dwErrorState.27 := bErrorNumber28;
dwErrorState.28 := bErrorNumber29;
dwErrorState.29 := bErrorNumber30;
dwErrorState.30 := bErrorNumber31;
dwErrorState.31 := bErrorNumber32;

(*-----------------------------------------------------------------------------------------------------------------------------------------------------------------------------------*)
(*Обрабатываем сброс флагов ошибок*)

RTRIGInst01(CLK := bErrorNumber01, Q => bErrorNumber01RTrig);
RTRIGInst02(CLK := bErrorNumber02, Q => bErrorNumber02RTrig);
RTRIGInst03(CLK := bErrorNumber03, Q => bErrorNumber03RTrig);
RTRIGInst04(CLK := bErrorNumber04, Q => bErrorNumber04RTrig);
RTRIGInst05(CLK := bErrorNumber05, Q => bErrorNumber05RTrig);
RTRIGInst06(CLK := bErrorNumber06, Q => bErrorNumber06RTrig);
RTRIGInst07(CLK := bErrorNumber07, Q => bErrorNumber07RTrig);
RTRIGInst08(CLK := bErrorNumber08, Q => bErrorNumber08RTrig);
RTRIGInst09(CLK := bErrorNumber09, Q => bErrorNumber09RTrig);
RTRIGInst10(CLK := bErrorNumber10, Q => bErrorNumber10RTrig);
RTRIGInst11(CLK := bErrorNumber11, Q => bErrorNumber11RTrig);
RTRIGInst12(CLK := bErrorNumber12, Q => bErrorNumber12RTrig);
RTRIGInst13(CLK := bErrorNumber13, Q => bErrorNumber13RTrig);
RTRIGInst14(CLK := bErrorNumber14, Q => bErrorNumber14RTrig);
RTRIGInst15(CLK := bErrorNumber15, Q => bErrorNumber15RTrig);
RTRIGInst16(CLK := bErrorNumber16, Q => bErrorNumber16RTrig);

RTRIGInst17(CLK := bErrorNumber17, Q => bErrorNumber17RTrig);
RTRIGInst18(CLK := bErrorNumber18, Q => bErrorNumber18RTrig);
RTRIGInst19(CLK := bErrorNumber19, Q => bErrorNumber19RTrig);
RTRIGInst20(CLK := bErrorNumber20, Q => bErrorNumber20RTrig);
RTRIGInst21(CLK := bErrorNumber21, Q => bErrorNumber21RTrig);
RTRIGInst22(CLK := bErrorNumber22, Q => bErrorNumber22RTrig);
RTRIGInst23(CLK := bErrorNumber23, Q => bErrorNumber23RTrig);
RTRIGInst24(CLK := bErrorNumber24, Q => bErrorNumber24RTrig);
RTRIGInst25(CLK := bErrorNumber25, Q => bErrorNumber25RTrig);
RTRIGInst26(CLK := bErrorNumber26, Q => bErrorNumber26RTrig);
RTRIGInst27(CLK := bErrorNumber27, Q => bErrorNumber27RTrig);
RTRIGInst28(CLK := bErrorNumber28, Q => bErrorNumber28RTrig);
RTRIGInst29(CLK := bErrorNumber29, Q => bErrorNumber29RTrig);
RTRIGInst30(CLK := bErrorNumber30, Q => bErrorNumber30RTrig);
RTRIGInst31(CLK := bErrorNumber31, Q => bErrorNumber31RTrig);
RTRIGInst32(CLK := bErrorNumber32, Q => bErrorNumber32RTrig);

RSInst01(SET := bErrorNumber01RTrig, RESET1 := bResetErrors, Q1 => bErrorNumber01Trig);
RSInst02(SET := bErrorNumber02RTrig, RESET1 := bResetErrors, Q1 => bErrorNumber02Trig);
RSInst03(SET := bErrorNumber03RTrig, RESET1 := bResetErrors, Q1 => bErrorNumber03Trig);
RSInst04(SET := bErrorNumber04RTrig, RESET1 := bResetErrors, Q1 => bErrorNumber04Trig);
RSInst05(SET := bErrorNumber05RTrig, RESET1 := bResetErrors, Q1 => bErrorNumber05Trig);
RSInst06(SET := bErrorNumber06RTrig, RESET1 := bResetErrors, Q1 => bErrorNumber06Trig);
RSInst07(SET := bErrorNumber07RTrig, RESET1 := bResetErrors, Q1 => bErrorNumber07Trig);
RSInst08(SET := bErrorNumber08RTrig, RESET1 := bResetErrors, Q1 => bErrorNumber08Trig);
RSInst09(SET := bErrorNumber09RTrig, RESET1 := bResetErrors, Q1 => bErrorNumber09Trig);
RSInst10(SET := bErrorNumber10RTrig, RESET1 := bResetErrors, Q1 => bErrorNumber10Trig);
RSInst11(SET := bErrorNumber11RTrig, RESET1 := bResetErrors, Q1 => bErrorNumber11Trig);
RSInst12(SET := bErrorNumber12RTrig, RESET1 := bResetErrors, Q1 => bErrorNumber12Trig);
RSInst13(SET := bErrorNumber13RTrig, RESET1 := bResetErrors, Q1 => bErrorNumber13Trig);
RSInst14(SET := bErrorNumber14RTrig, RESET1 := bResetErrors, Q1 => bErrorNumber14Trig);
RSInst15(SET := bErrorNumber15RTrig, RESET1 := bResetErrors, Q1 => bErrorNumber15Trig);
RSInst16(SET := bErrorNumber16RTrig, RESET1 := bResetErrors, Q1 => bErrorNumber16Trig);

RSInst17(SET := bErrorNumber17RTrig, RESET1 := bResetErrors, Q1 => bErrorNumber17Trig);
RSInst18(SET := bErrorNumber18RTrig, RESET1 := bResetErrors, Q1 => bErrorNumber18Trig);
RSInst19(SET := bErrorNumber19RTrig, RESET1 := bResetErrors, Q1 => bErrorNumber19Trig);
RSInst20(SET := bErrorNumber20RTrig, RESET1 := bResetErrors, Q1 => bErrorNumber20Trig);
RSInst21(SET := bErrorNumber21RTrig, RESET1 := bResetErrors, Q1 => bErrorNumber21Trig);
RSInst22(SET := bErrorNumber22RTrig, RESET1 := bResetErrors, Q1 => bErrorNumber22Trig);
RSInst23(SET := bErrorNumber23RTrig, RESET1 := bResetErrors, Q1 => bErrorNumber23Trig);
RSInst24(SET := bErrorNumber24RTrig, RESET1 := bResetErrors, Q1 => bErrorNumber24Trig);
RSInst25(SET := bErrorNumber25RTrig, RESET1 := bResetErrors, Q1 => bErrorNumber25Trig);
RSInst26(SET := bErrorNumber26RTrig, RESET1 := bResetErrors, Q1 => bErrorNumber26Trig);
RSInst27(SET := bErrorNumber27RTrig, RESET1 := bResetErrors, Q1 => bErrorNumber27Trig);
RSInst28(SET := bErrorNumber28RTrig, RESET1 := bResetErrors, Q1 => bErrorNumber28Trig);
RSInst29(SET := bErrorNumber29RTrig, RESET1 := bResetErrors, Q1 => bErrorNumber29Trig);
RSInst30(SET := bErrorNumber30RTrig, RESET1 := bResetErrors, Q1 => bErrorNumber30Trig);
RSInst31(SET := bErrorNumber31RTrig, RESET1 := bResetErrors, Q1 => bErrorNumber31Trig);
RSInst32(SET := bErrorNumber32RTrig, RESET1 := bResetErrors, Q1 => bErrorNumber32Trig);

bQX_Horn := (bErrorNumber01Trig OR
             (*bErrorNumber02Trig OR
             bErrorNumber03Trig OR*)
             bErrorNumber04Trig OR
             bErrorNumber05Trig OR
             bErrorNumber06Trig OR
             bErrorNumber07Trig OR
             bErrorNumber08Trig OR
             bErrorNumber09Trig OR
             bErrorNumber10Trig OR
             bErrorNumber11Trig OR
             bErrorNumber12Trig OR
             bErrorNumber13Trig OR
             bErrorNumber14Trig OR
             bErrorNumber15Trig OR
             bErrorNumber16Trig OR

			 bErrorNumber17Trig OR
             bErrorNumber18Trig OR
             bErrorNumber19Trig OR
             bErrorNumber20Trig OR
             bErrorNumber21Trig OR
             bErrorNumber22Trig OR
             bErrorNumber23Trig OR
             bErrorNumber24Trig OR
             bErrorNumber25Trig OR
             bErrorNumber26Trig OR
             bErrorNumber27Trig OR
             bErrorNumber28Trig OR
             bErrorNumber29Trig OR
 			 bErrorNumber30Trig OR
             bErrorNumber31Trig OR
             bErrorNumber32Trig);

(*-----------------------------------------------------------------------------------------------------------------------------------------------------------------------------------*)
(*Обрабатываем сброс флагов ошибок*)

IF bResetErrors = 1

THEN
	CAN1_WARNING   := 0;
	CAN1_BUSOFF    := 0;
	CAN2_WARNING   := 0;
	CAN2_BUSOFF    := 0;
(*	bErrorNumber01 := 0;
	bErrorNumber02 := 0;
	bErrorNumber03 := 0;*)
	bErrorNumber04 := 0;
	bErrorNumber05 := 0;
	bErrorNumber06 := 0;
	(*bErrorNumber07 := 0;*)
	bErrorNumber08 := 0;
	bErrorNumber09 := 0;
	(*bErrorNumber10 := 0;
	bErrorNumber11 := 0;
	bErrorNumber12 := 0;*)
	bErrorNumber13 := 0;
	bErrorNumber14 := 0;
	(*bErrorNumber15 := 0;
	bErrorNumber16 := 0;

	bErrorNumber17 := 0;
	bErrorNumber18 := 0;
	bErrorNumber19 := 0;*)
	bErrorNumber20 := 0;
	(*bErrorNumber21 := 0;
	bErrorNumber22 := 0;
	bErrorNumber23 := 0;
	bErrorNumber24 := 0;
	bErrorNumber25 := 0;*)
	bErrorNumber26 := 0;
	(*bErrorNumber27 := 0;
	bErrorNumber28 := 0;
	bErrorNumber29 := 0;
	bErrorNumber30 := 0;
	bErrorNumber31 := 0;
	bErrorNumber32 := 0:*)

END_IF;

(*-----------------------------------------------------------------------------------------------------------------------------------------------------------------------------------*)
(*Триггер на включение блокировки*)

RSInst(SET := NOT bQX_TriplexEmergStop, RESET1 := bResetErrors);
bQX_TriplexEmergStopTrig := NOT RSInst.Q1;

(*-----------------------------------------------------------------------------------------------------------------------------------------------------------------------------------*)
(**)

bResetErrors := 0;
END_PROGRAM

(* POU Output Modules/Horn_processing, ST *)
PROGRAM Horn_processing

VAR_INPUT
	bFirstIn    : BOOL;
END_VAR

VAR
	BLINK_HORN  : BLINK;
	bHornEnable : BOOL := 0;(**)
END_VAR
(*-----------------------------------------------------------------------------------------------------------------------------------------------------------------------------------*)
(**)

IF dwHornEnable <> 0
THEN
	bHornEnable := 1;
ELSE
	bHornEnable := 0;
END_IF;

BLINK_HORN(ENABLE := bHornEnable, TIMEHIGH := T#0.5S, TIMELOW := T#0.5S, OUT => bQX_Horn);
END_PROGRAM

(* POU Service/ServiceMeter_processing, ST *)
PROGRAM ServiceMeter_processing

VAR_INPUT
	bInit               : BOOL;
END_VAR

VAR
	bInitLocal          : BOOL := 1;
	ControllerTime      : TIMER_READ_US;
	dwTimeCurrent       : DWORD;
	dwTimePrevious      : DWORD;
	dwTime              : DWORD;

	instMemCpy          : MEMCPY;
	instFRAMWrite       : FRAMWRITE;
	instFRAMRead        : FRAMREAD;

	k                   : INT;
	i                   : INT;
END_VAR
(*-----------------------------------------------------------------------------------------------------------------------------------------------------------------------------------*)
(**)
(*
dwTotalServiceMeter := 3600;
instFRAMWrite(Enable := 1, DST := iMemAdrTotalServiceMeter, LEN := 4, SRC := ADR(dwTotalServiceMeter));
*)
(*-----------------------------------------------------------------------------------------------------------------------------------------------------------------------------------*)
(**)

IF bInit = 1
THEN
	instFRAMRead(Enable := 1, SRC := iMemAdrTotalServiceMeter, LEN := 4, DST := ADR(dwTotalServiceMeter));(*Первоначальное извлечение из FRAM значение моточасов*)
END_IF;

(*-----------------------------------------------------------------------------------------------------------------------------------------------------------------------------------*)
(*Считаем накопленное время раз в X циклов*)

IF k < 12_000 THEN k := k + 1; ELSE k := 0; END_IF;

IF k = 12_000
THEN

(*-----------------------------------------------------------------------------------------------------------------------------------------------------------------------------------*)
(*Берем текущее время контроллера*)

	ControllerTime(TIME_US => dwTimeCurrent);

	dwTime := (dwTimeCurrent - dwTimePrevious) / 1_000_000;

(*-----------------------------------------------------------------------------------------------------------------------------------------------------------------------------------*)
(*Суммируем время*)

	IF (*bInitLocal = 0 AND*) diCurrentEngineRPM > 100
	THEN
		instFRAMRead(Enable := 1, SRC := iMemAdrTotalServiceMeter, LEN := 4, DST := ADR(dwTotalServiceMeter));(*Извлечение из FRAM значение моточасов*)

		dwTotalServiceMeter := dwTotalServiceMeter + dwTime;(*Считаем суммарно наработанные моточасы*)
		dwLastServiceMeter  := dwLastServiceMeter  + dwTime;(*Считаем наработанные моточасы с последнего включения*)

		instFRAMWrite(Enable := 1, DST := iMemAdrTotalServiceMeter, LEN := 4, SRC := ADR(dwTotalServiceMeter)); (*Cохранение в FRAM значение моточасов*)
	END_IF;

(*-----------------------------------------------------------------------------------------------------------------------------------------------------------------------------------*)
(*Запоминаем текущее время контроллера для следующего цикла*)

	dwTimePrevious := dwTimeCurrent;

(*-----------------------------------------------------------------------------------------------------------------------------------------------------------------------------------*)
(*Переходим к следующему циклу*)
	bInitLocal := 0;

END_IF;

rTotalServiceMeterOut := DWORD_TO_REAL(REAL_TO_DWORD((DWORD_TO_REAL(dwTotalServiceMeter) / 60 / 60) * 10)) / 10;
rLastServiceMeterOut  := DWORD_TO_REAL(REAL_TO_DWORD((DWORD_TO_REAL(dwLastServiceMeter)  / 60 / 60) * 10)) / 10;

(*-----------------------------------------------------------------------------------------------------------------------------------------------------------------------------------*)
(**)
END_PROGRAM

(* POU DOUT_processing, ST *)
PROGRAM DOUT_processing

VAR_INPUT
	bInit         : BOOL;
END_VAR

VAR
END_VAR
(*-----------------------------------------------------------------------------------------------------------------------------------------------------------------------------------*)
(**)

IF bPressSensorRST = 1
THEN
	IF bErrorGN2_Pres = 0 AND rIW_GN2_Pres < 3
	THEN
		rWF_PresCor := rIW_GN2_Pres;
	END_IF;
END_IF;

bPressSensorRST := 0; (**)

(*-----------------------------------------------------------------------------------------------------------------------------------------------------------------------------------*)
(**)

dwOutputState := 16#0000;

dwOutputState.0  := bQX_TriplexEmergStopTrig (*bQX_TriplexEmergStop*);

dwOutputState.5  := bQX_Horn;
dwOutputState.6  := bQX_EngineStarterBlock;

dwOutputState.8  := bQX_TriplexRPMContrMode;
dwOutputState.9  := bQX_HydHeatPresContrMode;
dwOutputState.10 := bQX_BoostPresContrMode;

%QX0.11  := bQX_TriplexEmergStopTrig (*bQX_TriplexEmergStop*);     (*1-22*)

%QX1.4   := bQX_Horn;                 (*1-51*)
%QX1.0   := bQX_EngineStarterBlock;   (*1-48*)

%QX0.12  := bQX_TriplexRPMContrMode;  (*1-41*)
%QX0.13  := bQX_HydHeatPresContrMode; (*1-42*)
%QX0.14  := bQX_BoostPresContrMode;   (*1-43*)
END_PROGRAM
